// TIA Portal project "Pushbutton Control for Solenoid Operation" (V17)
// Pushbutton Control for Solenoid Operation
// When Switch 1 or Switch 2 (pushbuttons) is turned ON (pressed) and then turned OFF (released), then Solenoid will be ON.
// And then, when Switch 1 or Switch 2 (pushbuttons) are turned ON (pressed) and then turned OFF (released), then Solenoid will be OFF.

(* hardware
DEVICE "S7-1200 station_1"  S7-1200 Station
   slot 0: "Rack_0"  S7-1200 Rack  Rack  V1.0
   slot 1: "PLC_1"  CPU 1211C AC/DC/Rly  6ES7 211-1BE40-0XB0  V4.5
*)

// ===== PLC "PLC_1"  CPU 1211C AC/DC/Rly =====

VAR_GLOBAL   // PLC tag table "Default tag table"
   "Switch 1" AT %I0.0 : Bool;
   "Switch 2" AT %I0.1 : Bool;
   "Solenoid" AT %Q0.0 : Bool;
   "PB" AT %I0.2 : Bool;
   "Tag_1" AT %M0.0 : Bool;
   "Tag_2" AT %M0.1 : Bool;
   "Tag_3" AT %M0.2 : Bool;
END_VAR

ORGANIZATION_BLOCK "Main"   // OB1, LAD, ProgramCycle
TITLE = "Main Program Sweep (Cycle)"
{ S7_Optimized_Access := 'TRUE' }
VERSION : 0.1
   VAR_INPUT
      Initial_Call : Bool;   // Initial call of this OB
      Remanence : Bool;   // =True, if remanent data are available
   END_VAR
BEGIN

REGION Network 1
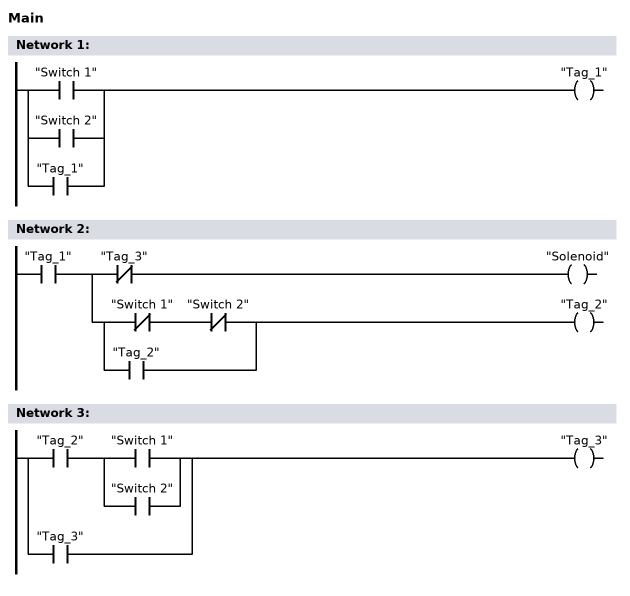
   RUNG wire#powerrail
      Contact( "Switch 1" )
      wire#w1
      Coil( "Tag_1" )
   END_RUNG
   RUNG wire#powerrail
      Contact( "Switch 2" )
   END_RUNG wire#w1
   RUNG wire#powerrail
      Contact( "Tag_1" )
   END_RUNG wire#w1
   // the same network as SCL:
   "Tag_1" := "Switch 1" OR "Switch 2" OR "Tag_1";
END_REGION

REGION Network 2
   RUNG wire#powerrail
      Contact( "Tag_1" )
      wire#w1
      I_Contact( "Tag_3" )
      Coil( "Solenoid" )
   END_RUNG
   RUNG wire#w1
      I_Contact( "Switch 1" )
      I_Contact( "Switch 2" )
      wire#w2
      Coil( "Tag_2" )
   END_RUNG
   RUNG wire#w1
      Contact( "Tag_2" )
   END_RUNG wire#w2
   // the same network as SCL:
   "Solenoid" := "Tag_1" AND NOT "Tag_3";
   "Tag_2" := "Tag_1" AND ((NOT "Switch 1" AND NOT "Switch 2") OR "Tag_2");
END_REGION

REGION Network 3
   RUNG wire#powerrail
      Contact( "Tag_2" )
      wire#w1
      Contact( "Switch 1" )
      wire#w2
      Coil( "Tag_3" )
   END_RUNG
   RUNG wire#w1
      Contact( "Switch 2" )
   END_RUNG wire#w2
   RUNG wire#powerrail
      Contact( "Tag_3" )
   END_RUNG wire#w2
   // the same network as SCL:
   "Tag_3" := ("Tag_2" AND ("Switch 1" OR "Switch 2")) OR "Tag_3";
END_REGION
END_ORGANIZATION_BLOCK